// SIMATIC S7-200 SMART project (STEP 7-Micro/WIN SMART), CPU SR40

SYMBOL_TABLE 表格 1
真空值              VD200
温度值              VD204
氮封值              VD208
罗茨启动真空设定         VD212
罗茨停机真空设定         VD216
温度报警设定           VD220
温度急停设定           VD224
目标真空             VD228
氮封压力报警设定         VD232
氮封压力急停设定         VD236
开启清洗电流设定         VW240
关闭清洗电流设定         VW242
开启吹扫电流设定         VW244
关闭吹扫电流设定         VW246
螺杆频率读取           VW100
螺杆电流读取           VW102
螺杆频率显示           VW104
螺杆电流显示           VW106
罗茨频率读取           VW108
罗茨电流读取           VW110
罗茨频率显示           VW112
罗茨电流显示           VW114
螺杆频率写入           VW116
罗茨频率写入           VW118
螺杆手动频率           VW120
罗茨手动频率           VW122
清洗时间设定           VW124
吹扫时间设定           VW126
清洗时间显示           VW128
吹扫时间显示           VW130
清洗时间中间量          VW132
吹扫时间中间量          VW134
自动步骤             VW20
延时定时器            T50
流量开关定时器          T51
清洗定时器            T37
吹扫定时器            T38
故障急停             V300.0
故障报警             V300.1
流量开关fault        V300.2
液位开关fault        V300.3
螺杆变频器fault       V300.4
罗茨变频器fault       V300.5
罗茨风机过载fault      V300.6
螺杆风机过载fault      V300.7
急停fault          V301.0
高温报警fault        V301.1
高温急停fault        V301.2
氮封过低报警fault      V301.3
氮封过低急停fault      V301.4
螺杆泵HMI           V500.0
罗茨泵HMI           V500.1
入口阀HMI           V500.2
清洗阀HMI           V500.3
吹扫阀HMI           V500.4
屏蔽蜂鸣器            V500.5
在线清洗HMI          V500.6
在线吹扫HMI          V500.7
END_SYMBOL_TABLE

SYMBOL_TABLE 系统符号
Always_On        SM0.0    // 始终接通
First_Scan_On    SM0.1    // 仅在第一个扫描周期时接通
Clock_1s         SM0.5    // 针对 1 s 的周期时间，时钟脉冲接通 0.5 s，断开 0.5 s.
END_SYMBOL_TABLE

SYMBOL_TABLE 表格 3
二读完成位            M2.3
二写完成位            M2.4
启动读写功            M0.1
通讯心跳             M11.2
延时触发             M30.0
一读完成位            M2.1
一写完成位            M2.2
主站错误代            MB1
主站完成位            M0.0
END_SYMBOL_TABLE

ORGANIZATION_BLOCK MAIN:OB1
TITLE=程序注释
BEGIN
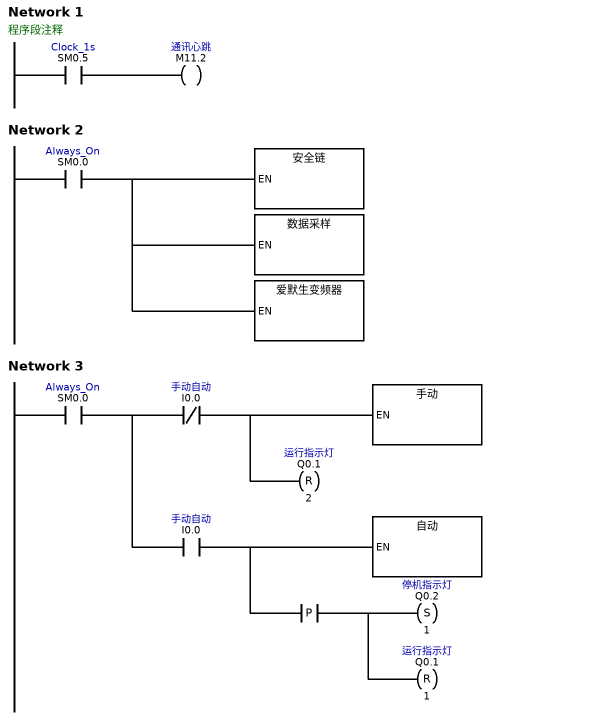
Network 1
// 程序段注释
LD     Clock_1s:SM0.5
=      通讯心跳:M11.2
Network 2
LD     Always_On:SM0.0
CALL   安全链:SBR2
CALL   数据采样:SBR1
CALL   爱默生变频器:SBR0
Network 3
LD     Always_On:SM0.0
LPS
AN     手动自动:I0.0
CALL   手动:SBR3
R      运行指示灯:Q0.1, 2
LPP
A      手动自动:I0.0
CALL   自动:SBR4
EU
S      停机指示灯:Q0.2, 1
R      运行指示灯:Q0.1, 1
END_ORGANIZATION_BLOCK

SUBROUTINE_BLOCK 爱默生变频器:SBR0
TITLE=子程序注释
BEGIN
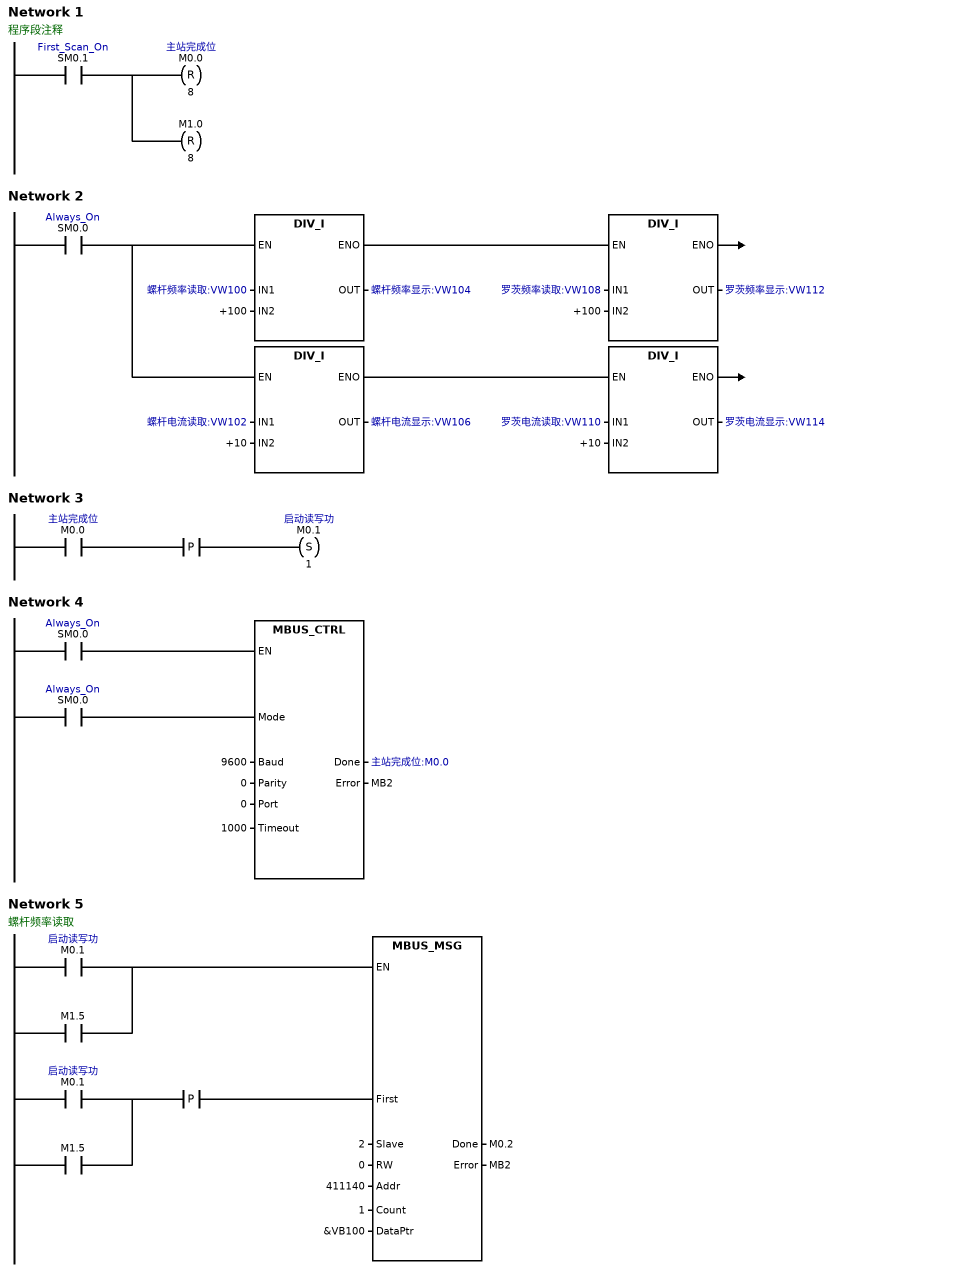
Network 1
// 程序段注释
LD     First_Scan_On:SM0.1
R      主站完成位:M0.0, 8
R      M1.0, 8
Network 2
LD     Always_On:SM0.0
LPS
MOVW   螺杆频率读取:VW100, 螺杆频率显示:VW104
AENO
/I     +100, 螺杆频率显示:VW104
AENO
MOVW   罗茨频率读取:VW108, 罗茨频率显示:VW112
/I     +100, 罗茨频率显示:VW112
LPP
MOVW   螺杆电流读取:VW102, 螺杆电流显示:VW106
AENO
/I     +10, 螺杆电流显示:VW106
AENO
MOVW   罗茨电流读取:VW110, 罗茨电流显示:VW114
/I     +10, 罗茨电流显示:VW114
Network 3
LD     主站完成位:M0.0
EU
S      启动读写功:M0.1, 1
Network 4
LD     Always_On:SM0.0
=      L60.0
LD     Always_On:SM0.0
=      L63.7
LD     L60.0
CALL   MBUS_CTRL:SBR7, L63.7, 9600, 0, 0, 1000, 主站完成位:M0.0, MB2
Network 5
// 螺杆频率读取
LD     启动读写功:M0.1
O      M1.5
=      L60.0
LD     启动读写功:M0.1
O      M1.5
EU
=      L63.7
LD     L60.0
CALL   MBUS_MSG:SBR8, L63.7, 2, 0, 411140, 1, &VB100, M0.2, MB2
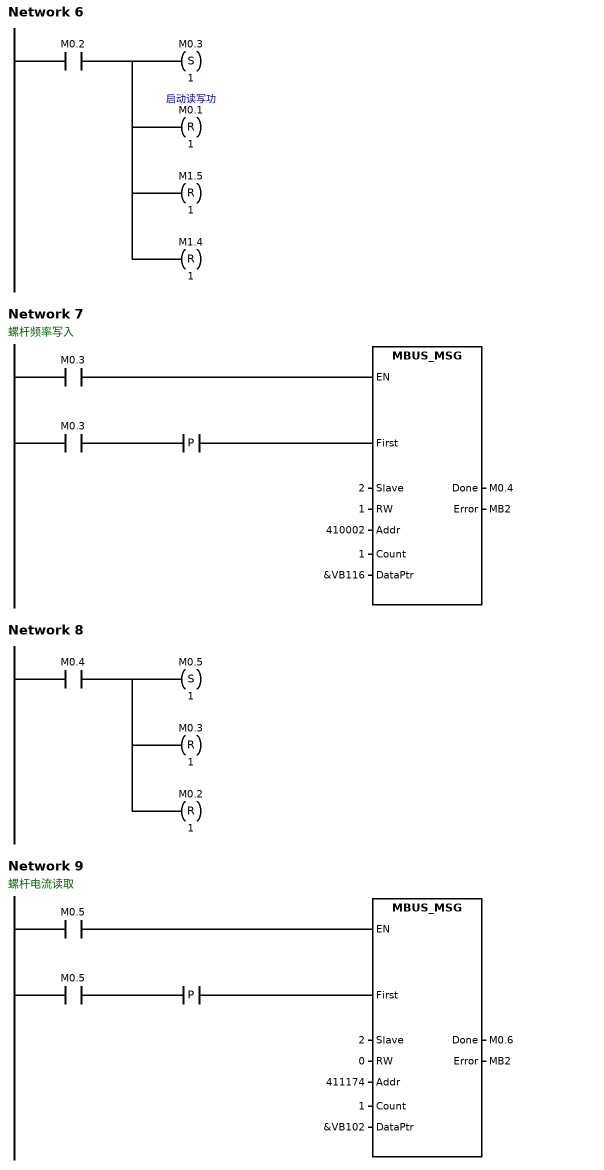
Network 6
LD     M0.2
S      M0.3, 1
R      启动读写功:M0.1, 1
R      M1.5, 1
R      M1.4, 1
Network 7
// 螺杆频率写入
LD     M0.3
=      L60.0
LD     M0.3
EU
=      L63.7
LD     L60.0
CALL   MBUS_MSG:SBR8, L63.7, 2, 1, 410002, 1, &VB116, M0.4, MB2
Network 8
LD     M0.4
S      M0.5, 1
R      M0.3, 1
R      M0.2, 1
Network 9
// 螺杆电流读取
LD     M0.5
=      L60.0
LD     M0.5
EU
=      L63.7
LD     L60.0
CALL   MBUS_MSG:SBR8, L63.7, 2, 0, 411174, 1, &VB102, M0.6, MB2
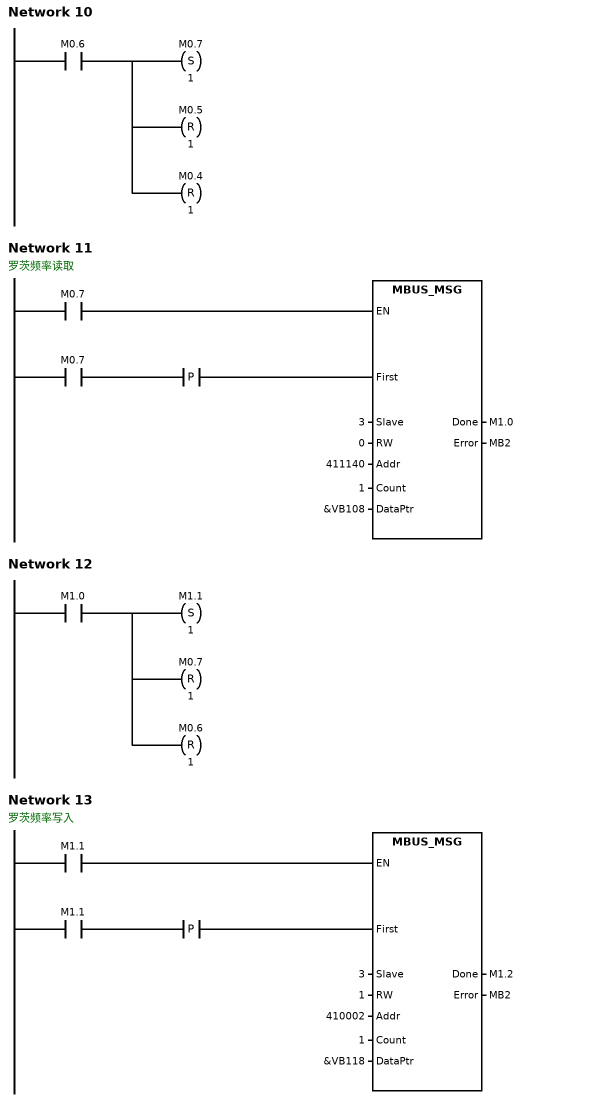
Network 10
LD     M0.6
S      M0.7, 1
R      M0.5, 1
R      M0.4, 1
Network 11
// 罗茨频率读取
LD     M0.7
=      L60.0
LD     M0.7
EU
=      L63.7
LD     L60.0
CALL   MBUS_MSG:SBR8, L63.7, 3, 0, 411140, 1, &VB108, M1.0, MB2
Network 12
LD     M1.0
S      M1.1, 1
R      M0.7, 1
R      M0.6, 1
Network 13
// 罗茨频率写入
LD     M1.1
=      L60.0
LD     M1.1
EU
=      L63.7
LD     L60.0
CALL   MBUS_MSG:SBR8, L63.7, 3, 1, 410002, 1, &VB118, M1.2, MB2
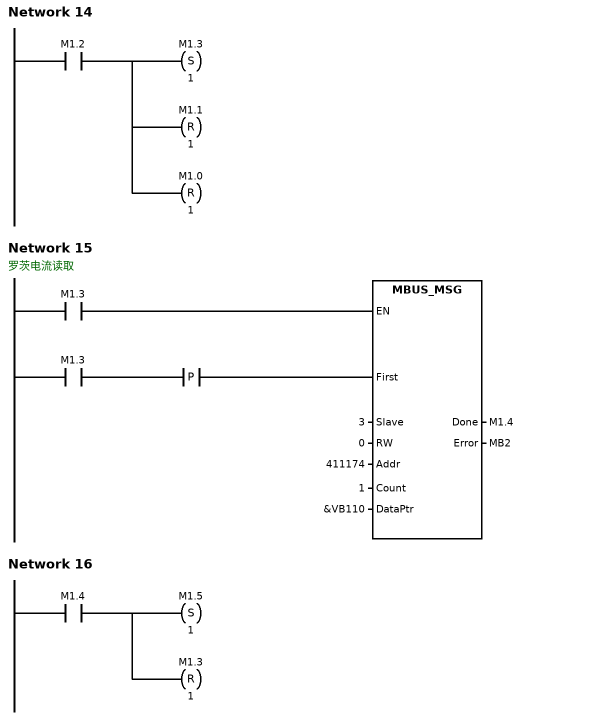
Network 14
LD     M1.2
S      M1.3, 1
R      M1.1, 1
R      M1.0, 1
Network 15
// 罗茨电流读取
LD     M1.3
=      L60.0
LD     M1.3
EU
=      L63.7
LD     L60.0
CALL   MBUS_MSG:SBR8, L63.7, 3, 0, 411174, 1, &VB110, M1.4, MB2
Network 16
LD     M1.4
S      M1.5, 1
R      M1.3, 1
END_SUBROUTINE_BLOCK

SUBROUTINE_BLOCK 数据采样:SBR1
TITLE=子程序注释
BEGIN
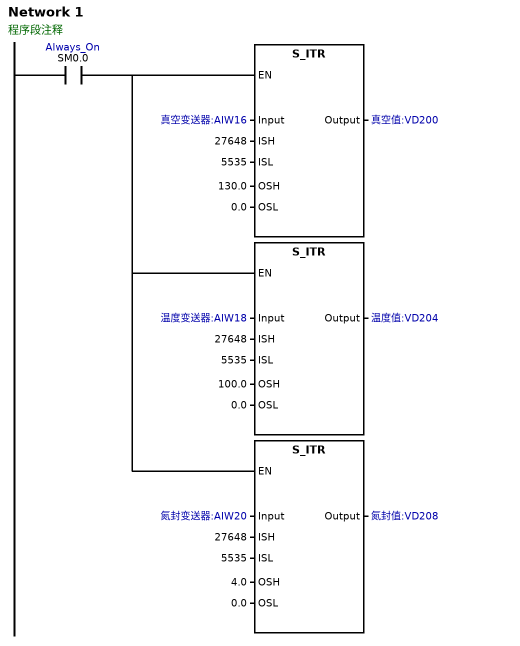
Network 1
// 程序段注释
LD     Always_On:SM0.0
CALL   S_ITR:SBR6, 真空变送器:AIW16, 27648, 5535, 130.0, 0.0, 真空值:VD200
CALL   S_ITR:SBR6, 温度变送器:AIW18, 27648, 5535, 100.0, 0.0, 温度值:VD204
CALL   S_ITR:SBR6, 氮封变送器:AIW20, 27648, 5535, 4.0, 0.0, 氮封值:VD208
END_SUBROUTINE_BLOCK

SUBROUTINE_BLOCK 安全链:SBR2
TITLE=子程序注释
BEGIN
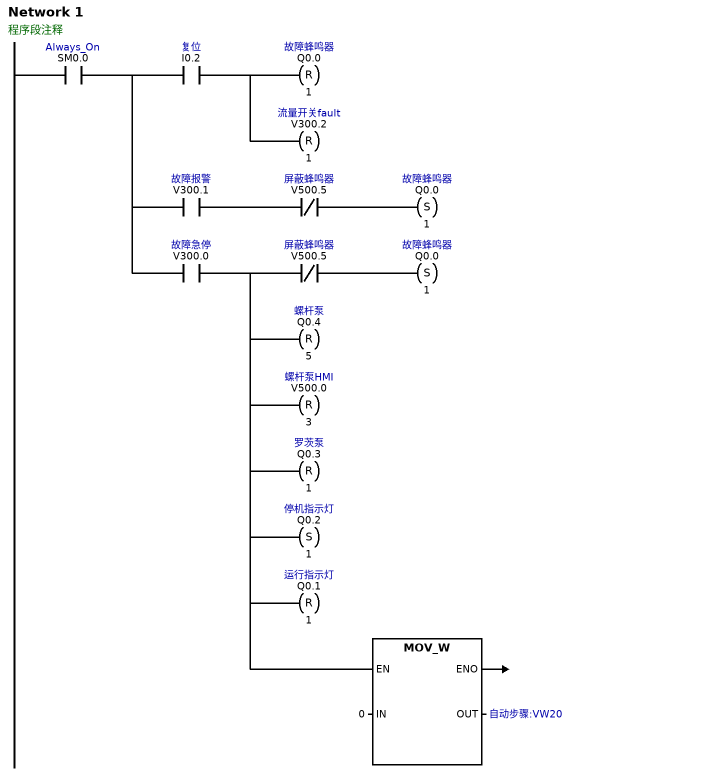
Network 1
// 程序段注释
LD     Always_On:SM0.0
LPS
A      复位:I0.2
R      故障蜂鸣器:Q0.0, 1
R      流量开关fault:V300.2, 1
LRD
A      故障报警:V300.1
AN     屏蔽蜂鸣器:V500.5
S      故障蜂鸣器:Q0.0, 1
LPP
A      故障急停:V300.0
LPS
AN     屏蔽蜂鸣器:V500.5
S      故障蜂鸣器:Q0.0, 1
LRD
R      螺杆泵:Q0.4, 5
LRD
R      螺杆泵HMI:V500.0, 3
LRD
R      罗茨泵:Q0.3, 1
LRD
S      停机指示灯:Q0.2, 1
LRD
R      运行指示灯:Q0.1, 1
LPP
MOVW   0, 自动步骤:VW20
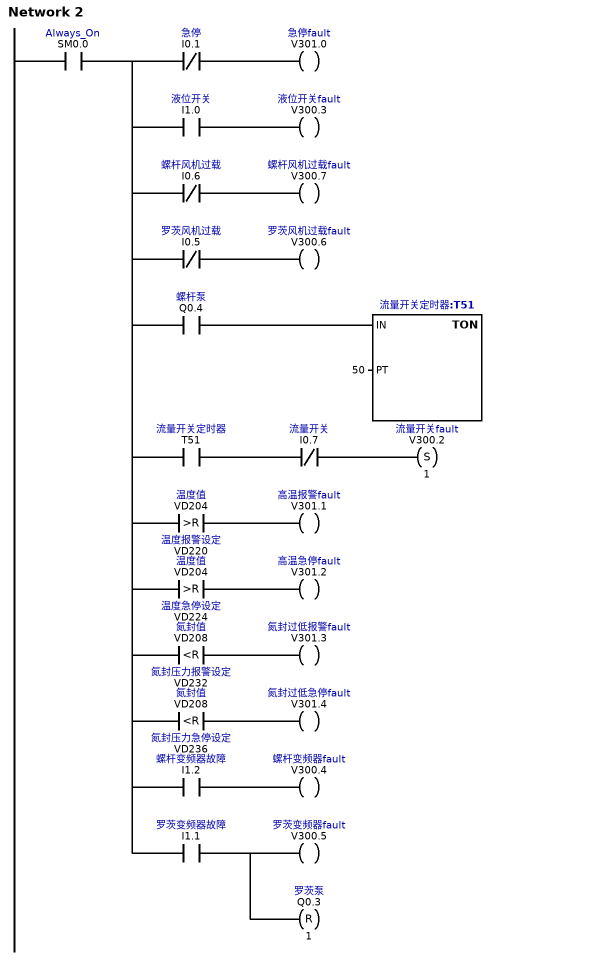
Network 2
LD     Always_On:SM0.0
LPS
AN     急停:I0.1
=      急停fault:V301.0
LRD
A      液位开关:I1.0
=      液位开关fault:V300.3
LRD
AN     螺杆风机过载:I0.6
=      螺杆风机过载fault:V300.7
LRD
AN     罗茨风机过载:I0.5
=      罗茨风机过载fault:V300.6
LRD
A      螺杆泵:Q0.4
TON    流量开关定时器:T51, 50
LRD
A      流量开关定时器:T51
AN     流量开关:I0.7
S      流量开关fault:V300.2, 1
LRD
AR>    温度值:VD204, 温度报警设定:VD220
=      高温报警fault:V301.1
LRD
AR>    温度值:VD204, 温度急停设定:VD224
=      高温急停fault:V301.2
LRD
AR<    氮封值:VD208, 氮封压力报警设定:VD232
=      氮封过低报警fault:V301.3
LRD
AR<    氮封值:VD208, 氮封压力急停设定:VD236
=      氮封过低急停fault:V301.4
LRD
A      螺杆变频器故障:I1.2
=      螺杆变频器fault:V300.4
LPP
A      罗茨变频器故障:I1.1
=      罗茨变频器fault:V300.5
R      罗茨泵:Q0.3, 1
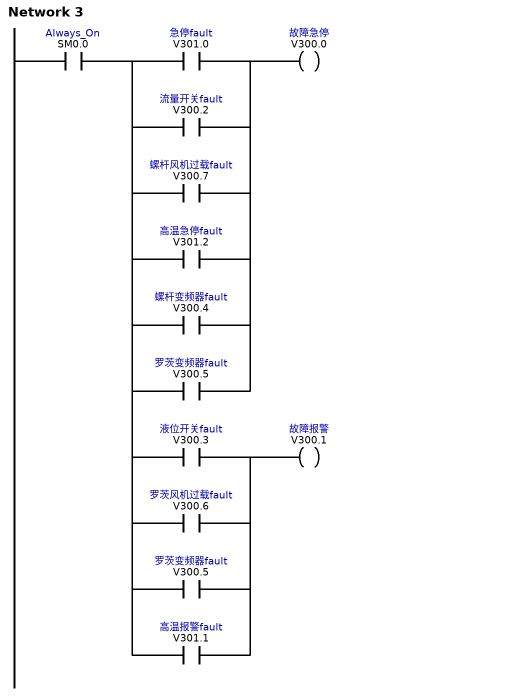
Network 3
LD     Always_On:SM0.0
LPS
LD     急停fault:V301.0
O      流量开关fault:V300.2
O      螺杆风机过载fault:V300.7
O      高温急停fault:V301.2
O      螺杆变频器fault:V300.4
O      罗茨变频器fault:V300.5
ALD
=      故障急停:V300.0
LPP
LD     液位开关fault:V300.3
O      罗茨风机过载fault:V300.6
O      罗茨变频器fault:V300.5
O      高温报警fault:V301.1
ALD
=      故障报警:V300.1
END_SUBROUTINE_BLOCK

SUBROUTINE_BLOCK 手动:SBR3
TITLE=子程序注释
BEGIN
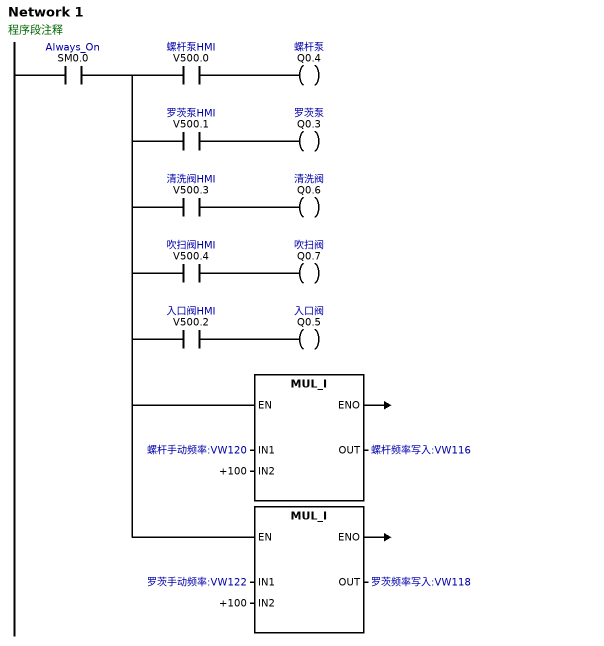
Network 1
// 程序段注释
LD     Always_On:SM0.0
LPS
A      螺杆泵HMI:V500.0
=      螺杆泵:Q0.4
LRD
A      罗茨泵HMI:V500.1
=      罗茨泵:Q0.3
LRD
A      清洗阀HMI:V500.3
=      清洗阀:Q0.6
LRD
A      吹扫阀HMI:V500.4
=      吹扫阀:Q0.7
LRD
A      入口阀HMI:V500.2
=      入口阀:Q0.5
LRD
MOVW   螺杆手动频率:VW120, 螺杆频率写入:VW116
*I     +100, 螺杆频率写入:VW116
LPP
MOVW   罗茨手动频率:VW122, 罗茨频率写入:VW118
*I     +100, 罗茨频率写入:VW118
END_SUBROUTINE_BLOCK

SUBROUTINE_BLOCK 自动:SBR4
TITLE=子程序注释
BEGIN
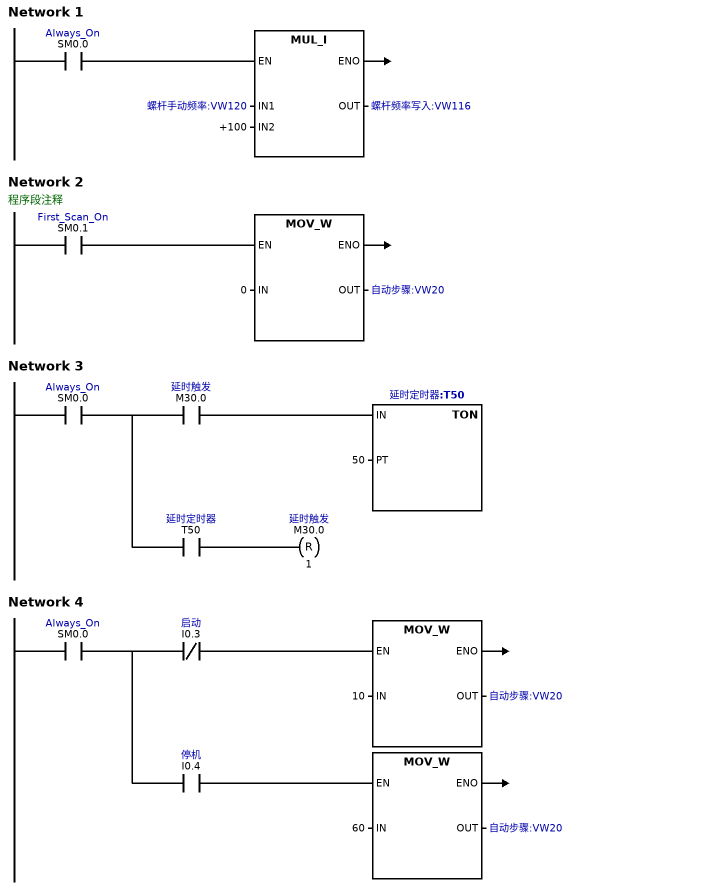
Network 1
LD     Always_On:SM0.0
MOVW   螺杆手动频率:VW120, 螺杆频率写入:VW116
*I     +100, 螺杆频率写入:VW116
Network 2
// 程序段注释
LD     First_Scan_On:SM0.1
MOVW   0, 自动步骤:VW20
Network 3
LD     Always_On:SM0.0
LPS
A      延时触发:M30.0
TON    延时定时器:T50, 50
LPP
A      延时定时器:T50
R      延时触发:M30.0, 1
Network 4
LD     Always_On:SM0.0
LPS
AN     启动:I0.3
MOVW   10, 自动步骤:VW20
LPP
A      停机:I0.4
MOVW   60, 自动步骤:VW20
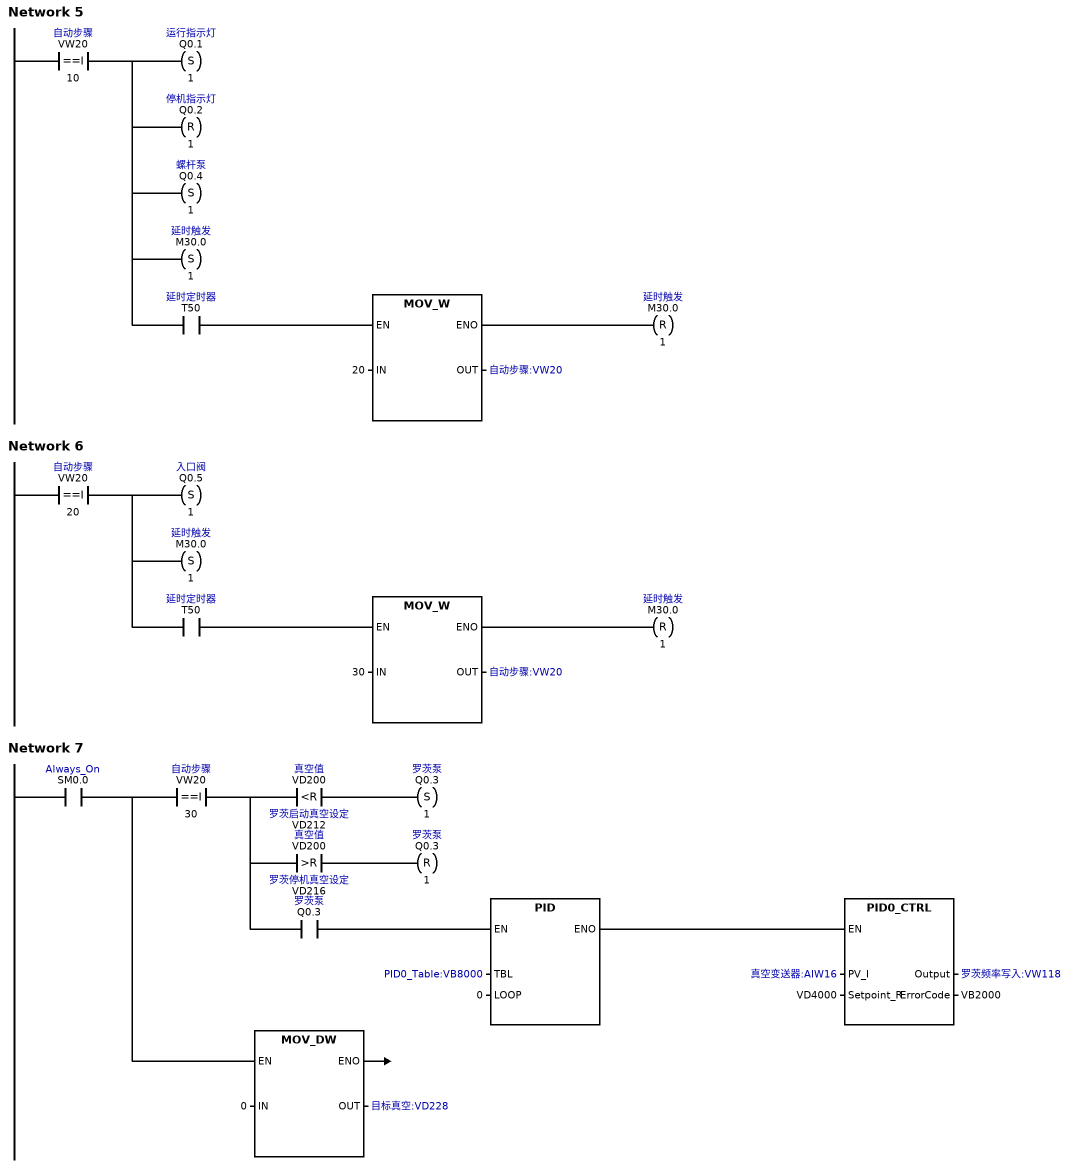
Network 5
LDW=   自动步骤:VW20, 10
S      运行指示灯:Q0.1, 1
R      停机指示灯:Q0.2, 1
S      螺杆泵:Q0.4, 1
S      延时触发:M30.0, 1
A      延时定时器:T50
MOVW   20, 自动步骤:VW20
AENO
R      延时触发:M30.0, 1
Network 6
LDW=   自动步骤:VW20, 20
S      入口阀:Q0.5, 1
S      延时触发:M30.0, 1
A      延时定时器:T50
MOVW   30, 自动步骤:VW20
AENO
R      延时触发:M30.0, 1
Network 7
LD     Always_On:SM0.0
LPS
AW=    自动步骤:VW20, 30
LPS
AR<    真空值:VD200, 罗茨启动真空设定:VD212
S      罗茨泵:Q0.3, 1
LRD
AR>    真空值:VD200, 罗茨停机真空设定:VD216
R      罗茨泵:Q0.3, 1
LPP
A      罗茨泵:Q0.3
PID    PID0_Table:VB8000, 0
AENO
CALL   PID0_CTRL:SBR5, 真空变送器:AIW16, VD4000, 罗茨频率写入:VW118, VB2000
LPP
MOVD   0, 目标真空:VD228
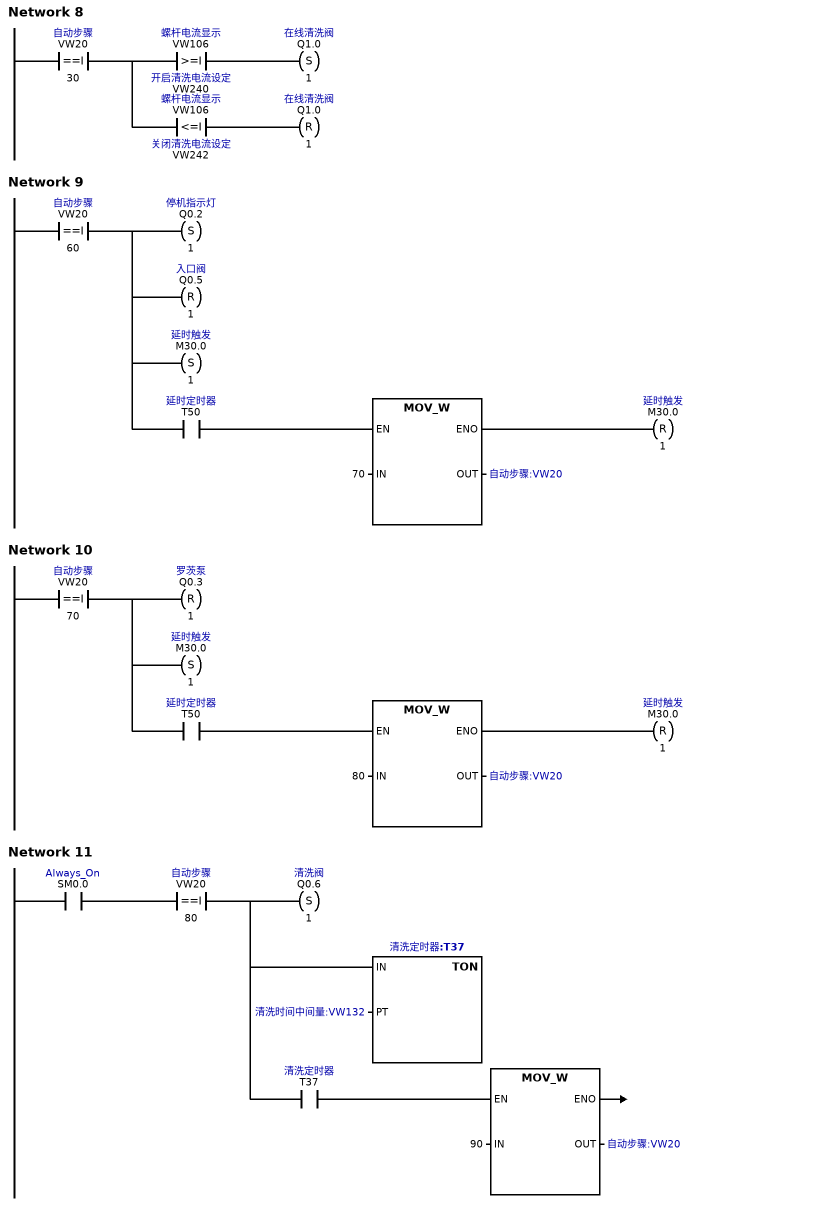
Network 8
LDW=   自动步骤:VW20, 30
LPS
AW>=   螺杆电流显示:VW106, 开启清洗电流设定:VW240
S      在线清洗阀:Q1.0, 1
LPP
AW<=   螺杆电流显示:VW106, 关闭清洗电流设定:VW242
R      在线清洗阀:Q1.0, 1
Network 9
LDW=   自动步骤:VW20, 60
S      停机指示灯:Q0.2, 1
R      入口阀:Q0.5, 1
S      延时触发:M30.0, 1
A      延时定时器:T50
MOVW   70, 自动步骤:VW20
AENO
R      延时触发:M30.0, 1
Network 10
LDW=   自动步骤:VW20, 70
R      罗茨泵:Q0.3, 1
S      延时触发:M30.0, 1
A      延时定时器:T50
MOVW   80, 自动步骤:VW20
AENO
R      延时触发:M30.0, 1
Network 11
LD     Always_On:SM0.0
AW=    自动步骤:VW20, 80
S      清洗阀:Q0.6, 1
TON    清洗定时器:T37, 清洗时间中间量:VW132
A      清洗定时器:T37
MOVW   90, 自动步骤:VW20
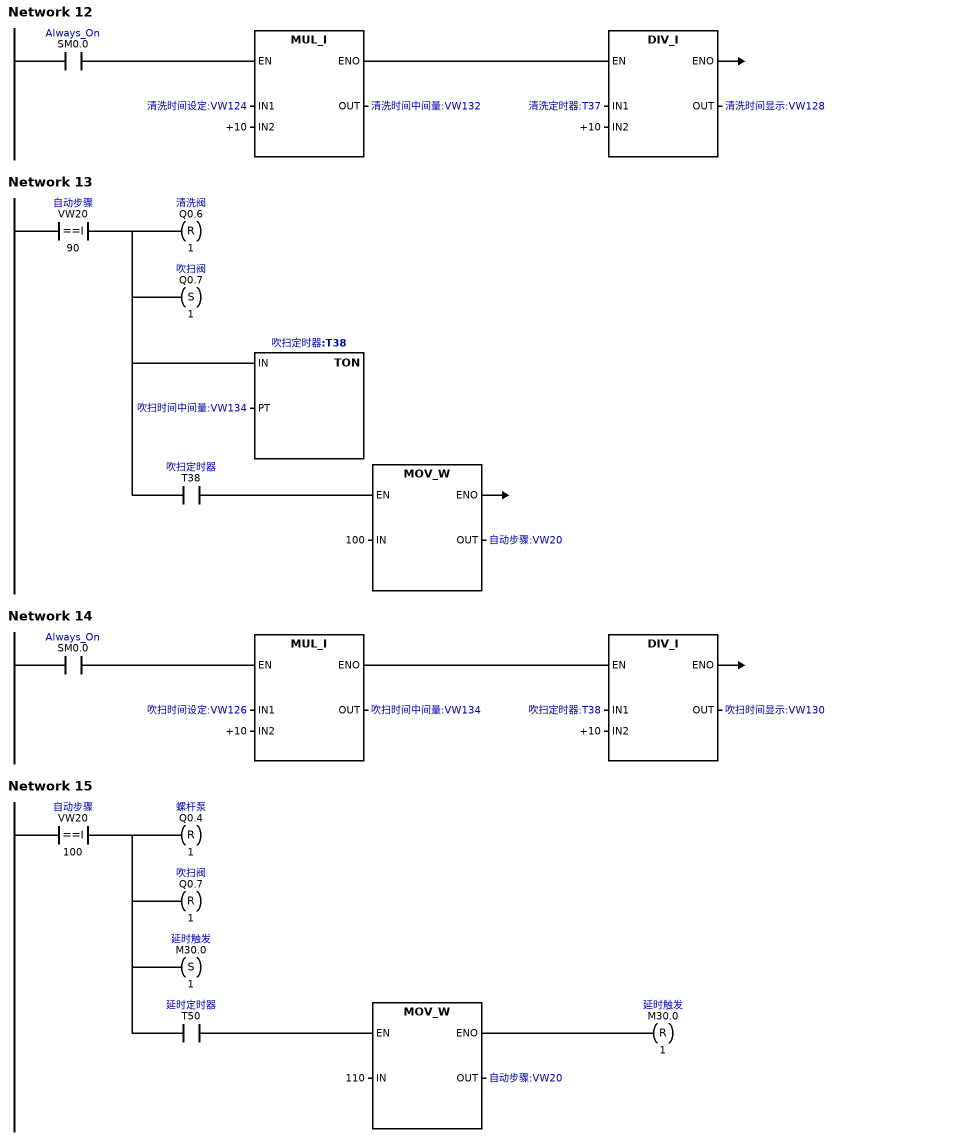
Network 12
LD     Always_On:SM0.0
MOVW   清洗时间设定:VW124, 清洗时间中间量:VW132
AENO
*I     +10, 清洗时间中间量:VW132
AENO
MOVW   清洗定时器:T37, 清洗时间显示:VW128
/I     +10, 清洗时间显示:VW128
Network 13
LDW=   自动步骤:VW20, 90
R      清洗阀:Q0.6, 1
S      吹扫阀:Q0.7, 1
TON    吹扫定时器:T38, 吹扫时间中间量:VW134
A      吹扫定时器:T38
MOVW   100, 自动步骤:VW20
Network 14
LD     Always_On:SM0.0
MOVW   吹扫时间设定:VW126, 吹扫时间中间量:VW134
AENO
*I     +10, 吹扫时间中间量:VW134
AENO
MOVW   吹扫定时器:T38, 吹扫时间显示:VW130
/I     +10, 吹扫时间显示:VW130
Network 15
LDW=   自动步骤:VW20, 100
R      螺杆泵:Q0.4, 1
R      吹扫阀:Q0.7, 1
S      延时触发:M30.0, 1
A      延时定时器:T50
MOVW   110, 自动步骤:VW20
AENO
R      延时触发:M30.0, 1
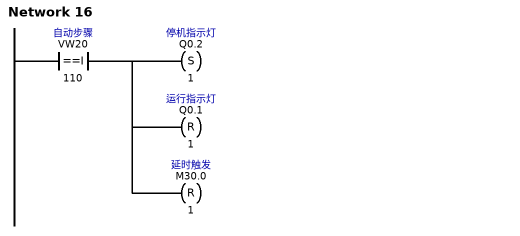
Network 16
LDW=   自动步骤:VW20, 110
S      停机指示灯:Q0.2, 1
R      运行指示灯:Q0.1, 1
R      延时触发:M30.0, 1
END_SUBROUTINE_BLOCK

// SBR5: protected block, not included

// SBR6: protected block, not included

// SBR7: protected block, not included

// SBR8: protected block, not included

// SBR9: protected block, not included

// SBR11: protected block, not included

// SBR12: protected block, not included

// SBR13: protected block, not included

// SBR14: protected block, not included

DATA_BLOCK_TAB 页面_1
BEGIN
//数据页注释
//按 F1 获取帮助和示例数据页
         罗茨启动真空设定, 6.0
         罗茨停机真空设定, 9.0
         温度报警设定, 45.0
         温度急停设定, 55.0
         目标真空, 0.0
         氮封压力报警设定, 0.0
         氮封压力急停设定, 0.0
         清洗时间设定, 300
         吹扫时间设定, 300
         螺杆手动频率, 50
         罗茨手动频率, 50
END_DATA_BLOCK_TAB
